INTERFACE I_Camera

METHOD ActivateCam : BOOL
VAR_INPUT
  iCameraSink : I_CameraSink;
END_VAR
END_METHOD

(*
  Activate/Deactivate camera trigger device
*)
PROPERTY bEnableTrigger : BOOL
SET
END_SET
END_PROPERTY

(*
  Activate/Deactivate camera manual teach mode
*)
PROPERTY bManualTeach : BOOL
SET
END_SET
END_PROPERTY

{attribute 'monitoring':='call'}
PROPERTY bSimulate : BOOL
GET
END_GET
SET
END_SET
END_PROPERTY

METHOD DeactivateCam : BOOL
VAR_INPUT
  iSink : I_CameraSink;
END_VAR
END_METHOD

{attribute 'monitoring':='call'}
PROPERTY ABSTRACT eCameraMode : E_CameraMode
GET
END_GET
END_PROPERTY

{attribute 'monitoring':='call'}
PROPERTY ABSTRACT eDeviceType : E_CameraDevice
GET
END_GET
END_PROPERTY

{attribute 'monitoring':='call'}
PROPERTY fCameraToPrintOffset : LREAL
GET
END_GET
END_PROPERTY

{attribute 'monitoring':='call'}
PROPERTY fDetectToCameraOffset : LREAL
GET
END_GET
END_PROPERTY

{attribute 'monitoring':='call'}
// camera frame size in [px]
PROPERTY fFrameLength : LREAL
GET
END_GET
SET
END_SET
END_PROPERTY

{attribute 'monitoring':='call'}
(*Image Length/Depth in [m]*)
PROPERTY fImageLength : LREAL
GET
END_GET
SET
END_SET
END_PROPERTY

{attribute 'monitoring':='call'}
(*Image Width in [m]*)
PROPERTY fImageWidth : LREAL
GET
END_GET
SET
END_SET
END_PROPERTY

{attribute 'monitoring':='call'}
(*Substrate Length/Depth in [m]*)
PROPERTY fSubstrateLength : LREAL
GET
END_GET
SET
END_SET
END_PROPERTY

{attribute 'monitoring':='call'}
(*Substrate Width in [m]*)
PROPERTY fSubstrateWidth : LREAL
GET
END_GET
SET
END_SET
END_PROPERTY

{attribute 'monitoring':='call'}
PROPERTY fTriggerDistance : LREAL
GET
END_GET
SET
END_SET
END_PROPERTY

(*
  Get camera status.
  :return: TRUE if camera is ok
*)
METHOD GetCamStatus : BOOL  // Camera Ok?
VAR_OUTPUT
  bConnectionOK  : BOOL;    // Camera connected
  bTeachOk       : BOOL;    // Teach successful
  nTeachedPoints : UDINT;   // Teached points for this job
  nScannedPoints : UDINT;   // Scanned points on current CT
  bCamStarted    : BOOL;    // Camera trigger is active, cam started
  bCamDone       : BOOL;    // Camera finished on last CT
  bErrors        : ARRAY[1..GVL_Camera.nC_NbCamErrors] OF BOOL;  // generic error flag list
END_VAR
END_METHOD

METHOD mJobStart : BOOL
VAR_INPUT
END_VAR
END_METHOD

(*
  Set mode to camera.
  :return: TRUE if success
*)
METHOD setCameraMode : BOOL
VAR_INPUT
  eCameraMode : E_CameraMode;
END_VAR
END_METHOD

METHOD setMsgInterface : BOOL
VAR_INPUT
  pMsgConfig  : POINTER TO ST_MSG_CONFIG;
END_VAR
END_METHOD

{attribute 'monitoring':='call'}
PROPERTY sName : STRING
GET
END_GET
END_PROPERTY

{attribute 'monitoring':='call'}
PROPERTY sVisuName : STRING
GET
END_GET
END_PROPERTY

END_INTERFACE

(* stored: Version 1.1.0.1, ProductVersion 3.1.4024.3
   Itf I_Camera: Id {5674f1fe-9d4a-41a3-a0a1-c185e43bbf40}
   Method ActivateCam: Id {ba8412d7-fb53-486a-94f9-8b39464fac5a}
   Property bEnableTrigger: Id {a64c3322-bafe-4f67-8776-8ae6263c1ac8}
   Set Set: Id {3b90e5d6-9ab2-4fa1-a22c-1e1c282db57e}
   Property bManualTeach: Id {6b655c17-33fd-48f5-9dbb-b18f90bf2b24}
   Set Set: Id {4ee6f514-8b64-449a-9cdf-700830169291}
   Property bSimulate: Id {ecf625f3-c312-45c3-a7f0-ac2547d849ba}
   Get Get: Id {d453bc16-cc12-495d-8cb5-2da1b606a550}
   Set Set: Id {4b8d8805-45c4-4ce2-abaf-786b8b61bbc6}
   Method DeactivateCam: Id {7d5fa3a8-e3d0-41e7-bd31-4eeb5568fecb}
   Property eCameraMode: Id {8faaf914-9316-4c9f-83cd-5dd71de4ce9d}
   Get Get: Id {c20daac4-cc1b-428c-8898-93d4ee00fe19}
   Property eDeviceType: Id {4df248e0-2e60-4bb3-a577-249a851b1fba}
   Get Get: Id {c7914735-d194-4368-9f36-4e8f60194ad2}
   Property fCameraToPrintOffset: Id {b8f23e9c-b746-4eae-9181-55a641350b9c}
   Get Get: Id {f24208cb-800c-4676-bb1c-78d12da77147}
   Property fDetectToCameraOffset: Id {fc74ba70-acb5-4a0c-a7e2-2783838252ba}
   Get Get: Id {9216a060-21d3-4813-85d2-c6a3d5ec6c74}
   Property fFrameLength: Id {ade4c057-e69d-43c6-83f5-d359e7abdf22}
   Get Get: Id {2ebc9aa7-4f34-41e5-a600-f390699dc3d9}
   Set Set: Id {799d7ea2-bfaa-404a-936b-12c5761c6043}
   Property fImageLength: Id {e64a7258-3e71-42ce-9230-29b5bd147720}
   Get Get: Id {cc6abbc8-10c2-406c-a539-d34315de89d3}
   Set Set: Id {76cb80cd-0523-4cbc-83b5-ca3c2d845ebd}
   Property fImageWidth: Id {354223c6-e242-498f-aa8d-a6b74a7d0eb5}
   Get Get: Id {fcb301de-810e-4eed-87cd-8eae68e11e78}
   Set Set: Id {61d153e2-ded1-40e2-a791-744c4461b95d}
   Property fSubstrateLength: Id {56a175eb-4401-420e-9500-315d7219a34e}
   Get Get: Id {cceed54b-87ae-446f-a107-0a624e9b91fd}
   Set Set: Id {35cd2beb-136f-41c0-9e7d-222824614ee2}
   Property fSubstrateWidth: Id {0a116a87-5d7a-4767-b42c-5b31dfac99a6}
   Get Get: Id {5d9c0a2a-1ad7-4537-bfc7-46fe3e65c97a}
   Set Set: Id {295bfefd-fa04-499b-a128-06477271140c}
   Property fTriggerDistance: Id {355820a8-6dbe-4bcf-9b87-5d8005bff447}
   Get Get: Id {a1e53b95-83c1-44fa-bfbf-3d57b21718ea}
   Set Set: Id {14176d0c-d6e0-4ae0-9bee-95877fc7a6dc}
   Method GetCamStatus: Id {4b1b0162-d8c5-4a44-9473-4479f539f751}
   Method mJobStart: Id {07d1a74f-9c1e-4b4b-8bfb-4ff2a66ef044}
   Method setCameraMode: Id {2bb20ac8-ea6c-4563-8a6d-3e931984b23d}
   Method setMsgInterface: Id {15efc3f9-e69e-49f3-9b43-1bb165d34029}
   Property sName: Id {1c9c1a68-ccc5-4476-a9cb-354759a69d5f}
   Get Get: Id {9acf0ac1-4aff-4e1f-a321-8d546aa70145}
   Property sVisuName: Id {6445ae93-9c91-4e6d-b53c-d90de3357d5c}
   Get Get: Id {81275749-1a4d-488d-aeda-04f764a44099} *)
